FUNCTION_BLOCK FB_SimpleRotaryTwoWayDrive EXTENDS FB_Unit
VAR_INPUT
END_VAR
VAR_OUTPUT
END_VAR
VAR
END_VAR

END_FUNCTION_BLOCK

(* stored: Version 1.1.0.1, ProductVersion 3.1.4024.11
   POU FB_SimpleRotaryTwoWayDrive: Id {91ccde8e-c8b2-4c10-8627-24b2c55efbe7}, SpecialFunc None *)
